// TIA Portal V18 export
FUNCTION_BLOCK "shiftTrigger"   // FB4, FBD
{ S7_Optimized_Access := 'TRUE' }
// stored: MemoryReserve 100, SetENOAutomatically false
   VAR_INPUT
      autostartEnabled { ExternalAccessible := 'False'; ExternalVisible := 'False'; ExternalWritable := 'False'} : Bool;
      actualTOD { ExternalAccessible := 'False'; ExternalVisible := 'False'; ExternalWritable := 'False'} : Time_Of_Day;
      actualDTL : DTL;
      shiftSettings { ExternalAccessible := 'False'; ExternalVisible := 'False'; ExternalWritable := 'False'} : "UDT_settingsShift";
   END_VAR
   VAR_OUTPUT
      active : Bool;
      taktTimeEn { ExternalAccessible := 'False'; ExternalVisible := 'False'; ExternalWritable := 'False'} : Bool;
      edgeShiftStartDetect { ExternalAccessible := 'False'; ExternalVisible := 'False'; ExternalWritable := 'False'} : Bool;
   END_VAR
   VAR
      P_edgeShiftStartDetect : Bool;
   END_VAR
   VAR_TEMP
      T_shiftActive : Bool;
      T_break1Active : Bool;
      T_break2Active : Bool;
      T_break3Active : Bool;
      T_break4Active : Bool;
      T_break5Active : Bool;
      T_endShiftStartDetect : Time_Of_Day;
      T_ShiftStartDetect : Bool;
   END_VAR
   VAR_TEMP   // added for the SCL form of the ladder/FBD networks
      _w1 : Bool;
   END_VAR
BEGIN

REGION Network 1: Settings shift EN / Shift trigger disabled
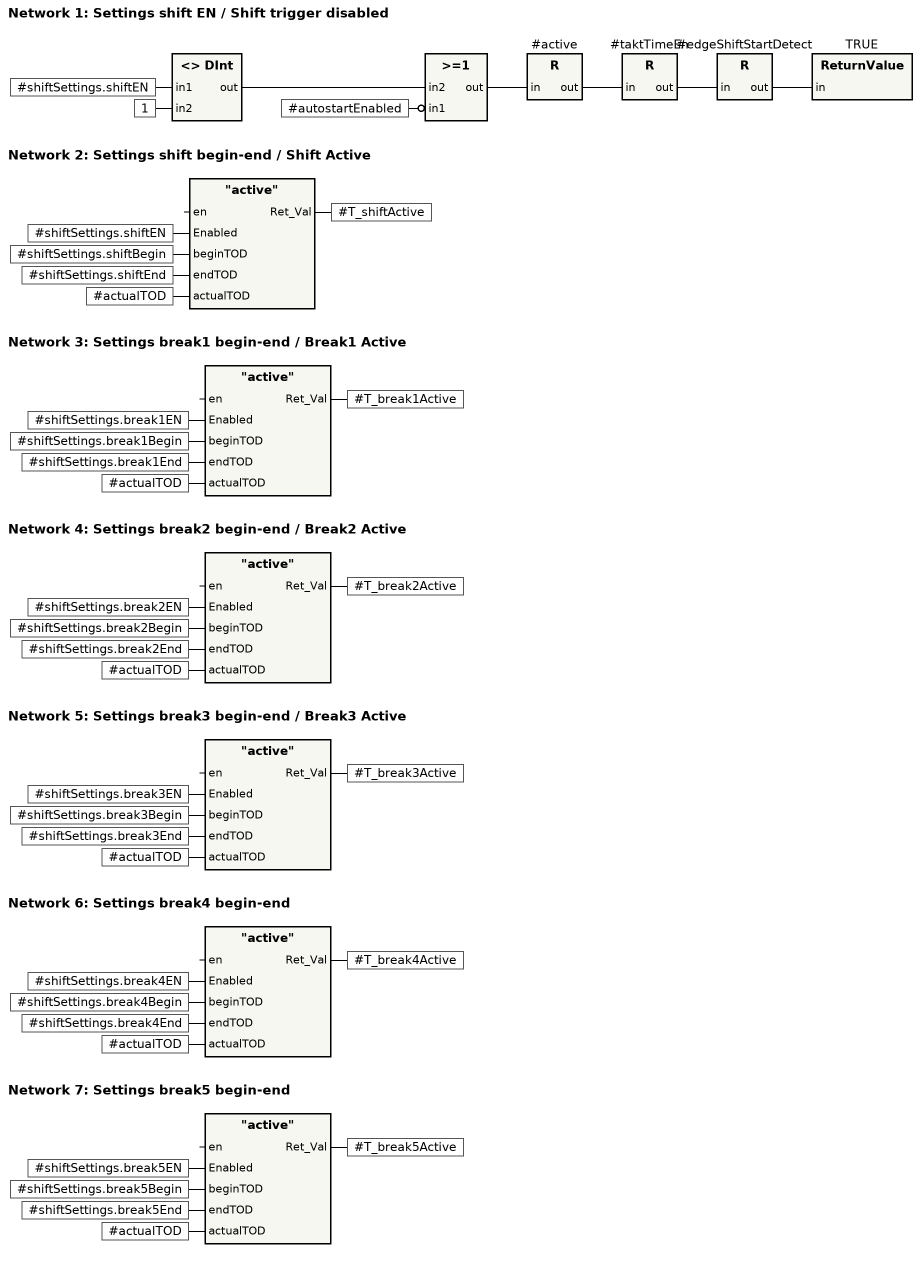
   #_w1 := (#shiftSettings.shiftEN <> 1) OR NOT #autostartEnabled;
   IF #_w1 THEN
       #active := FALSE;
       #taktTimeEn := FALSE;
       #edgeShiftStartDetect := FALSE;
       ENO := TRUE;
       RETURN;
   END_IF;
END_REGION

REGION Network 2: Settings shift begin-end / Shift Active
   #T_shiftActive := "active"(Enabled := #shiftSettings.shiftEN,
                           beginTOD := #shiftSettings.shiftBegin,
                           endTOD := #shiftSettings.shiftEnd,
                           actualTOD := #actualTOD);
END_REGION

REGION Network 3: Settings break1 begin-end / Break1 Active
   #T_break1Active := "active"(Enabled := #shiftSettings.break1EN,
                           beginTOD := #shiftSettings.break1Begin,
                           endTOD := #shiftSettings.break1End,
                           actualTOD := #actualTOD);
END_REGION

REGION Network 4: Settings break2 begin-end / Break2 Active
   #T_break2Active := "active"(Enabled := #shiftSettings.break2EN,
                           beginTOD := #shiftSettings.break2Begin,
                           endTOD := #shiftSettings.break2End,
                           actualTOD := #actualTOD);
END_REGION

REGION Network 5: Settings break3 begin-end / Break3 Active
   #T_break3Active := "active"(Enabled := #shiftSettings.break3EN,
                           beginTOD := #shiftSettings.break3Begin,
                           endTOD := #shiftSettings.break3End,
                           actualTOD := #actualTOD);
END_REGION

REGION Network 6: Settings break4 begin-end
   #T_break4Active := "active"(Enabled := #shiftSettings.break4EN,
                           beginTOD := #shiftSettings.break4Begin,
                           endTOD := #shiftSettings.break4End,
                           actualTOD := #actualTOD);
END_REGION

REGION Network 7: Settings break5 begin-end
   #T_break5Active := "active"(Enabled := #shiftSettings.break5EN,
                           beginTOD := #shiftSettings.break5Begin,
                           endTOD := #shiftSettings.break5End,
                           actualTOD := #actualTOD);
END_REGION

REGION Network 8: shift start detect signal duration
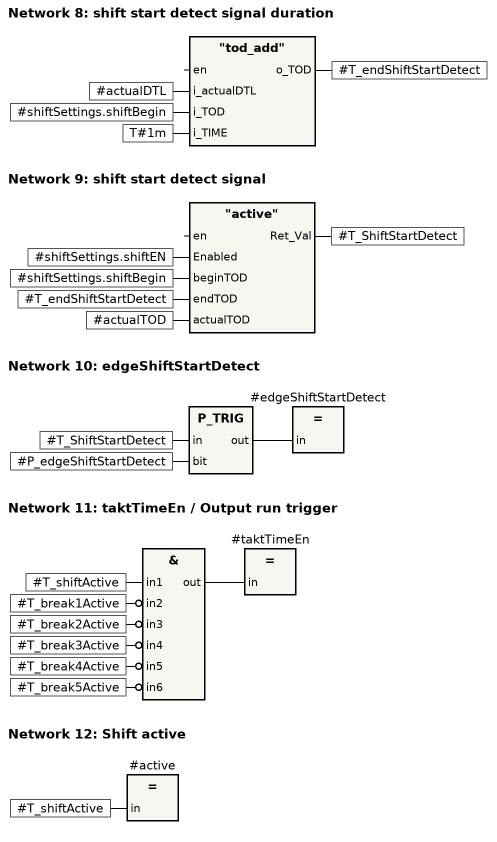
   "tod_add"(i_actualDTL := #actualDTL,
             i_TOD := #shiftSettings.shiftBegin,
             i_TIME := T#1m,
             o_TOD => #T_endShiftStartDetect);
END_REGION

REGION Network 9: shift start detect signal
   #T_ShiftStartDetect := "active"(Enabled := #shiftSettings.shiftEN,
                           beginTOD := #shiftSettings.shiftBegin,
                           endTOD := #T_endShiftStartDetect,
                           actualTOD := #actualTOD);
END_REGION

REGION Network 10: edgeShiftStartDetect
   #_w1 := #T_ShiftStartDetect AND NOT #P_edgeShiftStartDetect;   // rising edge
   #P_edgeShiftStartDetect := #T_ShiftStartDetect;
   #edgeShiftStartDetect := #_w1;
END_REGION

REGION Network 11: taktTimeEn / Output run trigger
   #taktTimeEn := #T_shiftActive AND NOT #T_break1Active AND NOT #T_break2Active AND NOT #T_break3Active AND NOT #T_break4Active AND NOT #T_break5Active;
END_REGION

REGION Network 12: Shift active
   #active := #T_shiftActive;
END_REGION
END_FUNCTION_BLOCK
